FUNCTION_BLOCK FB_SPECIAL_2
VAR_INPUT
	IN : 	BOOL;
	Run :	BOOL;		//Emitter = Run
	SpawnAmount : INT := 2;
//	Sensor : BOOL;		//mieluummin käytän ei sensoriin liittyvän ratkaisun
END_VAR
VAR_OUTPUT
	Q :			BOOL;
	Emitter : 	BOOL;	//Emitter = Run
	Remover :	BOOL;	//Remover = Run
END_VAR
VAR
	iState: INT;
	fbTON: TON;
	fbTON2: TON;
	X0: BOOL;
	i: INT;
END_VAR

IF NOT IN THEN
	Q := FALSE;
	iState := 0;
	ELSE
		Q := TRUE;
	//	Emitter := Run;		//Toimi ihan hyvin kun 1 kpl riittää
		Remover := Run;		
END_IF

IF Run = TRUE AND X0 = FALSE THEN
	X0 := TRUE;
END_IF

//äh, for-loopin tein ja se varmaan toimiki mutta aivan muualla oli bugi
//kuten myös R_TRIGulla olis kannattanu... meni jo
IF X0 AND i < SpawnAmount THEN			//1s välein väläyttää Emitteriä SpawnAmountin verran (3 oletus)
	fbTON(IN := TRUE, PT := T#2000MS);
	IF fbTON.Q THEN
		Emitter := TRUE;
		fbTON2(IN:=TRUE, PT := T#100MS);
		IF fbTON2.Q THEN
			Emitter := FALSE;
			fbTON2(IN := FALSE);
			fbTON(IN := FALSE);
			i := i+1;
		END_IF
	END_IF
ELSE 
	X0 := 		FALSE;
	Emitter := 	FALSE;
	i := 		0;
END_IF

END_FUNCTION_BLOCK

(* stored: Version 1.1.0.1, ProductVersion 3.1.4024.6
   POU FB_SPECIAL_2: Id {9734b71b-74ab-487c-85af-c68c3f7b38ab}, SpecialFunc None *)
